(* IEC 61131-3 sources: eCockpitGit/test_project/src/%F%00 Library/%F%JSON/%POU%FB_JSONWriter, 3 files *)

(* ---- %METH%deinitialize.st ---- *)
// |**Version**|**Author**| **Date** |**Changes**
// | 1         | NSN      | 22-06-20 | Creation
METHOD deinitialize

(*%!%__DELIMITER__%!%*)
IF ready THEN
	//Closes up remaining structs
	WHILE treeLevel > 0 DO
		CASE treeTypes[treeLevel] OF
			EStructType.object,EStructType.tArray:
				structEnd();
		END_CASE
	END_WHILE
	bufferPosition			:=		bufferPosition - 1;
	bufferPosition^			:=		EASCII.Null;
	//Initialisation is done
	ready					:=		FALSE;
	//Values are reset
	bufferMaxADR			:=		0;
	inArray					:=		FALSE;
	inObject				:=		FALSE;
	singleVal				:=		FALSE;
	lastComma				:=		0;
	bottomTypeInt			:=		EStructType.none;
	treeLevel				:=		0;
END_IF

(* ---- %METH%initialize.st ---- *)
//This initializes the manager with the correct values
// |**Version**|**Author**| **Date** |**Changes**
// | 1         | NSN      | 22-06-20 | Creation
METHOD initialize : SLMResult
VAR_INPUT
	buffer			:POINTER TO BYTE;	//The address of the file buffer
	bufferSize		:DWORD;				//The size of the file buffer
	singleLine		:BOOL;
	bottomType		:EStructType;
END_VAR
(*%!%__DELIMITER__%!%*)
//Buffer ADR is recorded
IF NOT(ready) THEN
	IF buffer <> 0 AND bufferSize <> 0 THEN
		bufferPosition		:=		buffer;
		bufferAddress		:=		buffer;
		bufferMaxADR		:=		bufferPosition + bufferSize;
		useSingleLine		:=		singleLine;
		bufferInvalid		:=		FALSE;
		//Initialisation is done
		ready				:=		TRUE;
		//First curly bracket is added
		bottomTypeInt		:=		bottomType;
		CASE bottomType OF
			EStructType.object:
				afterKey	:=		TRUE;
				objectStart(singleLine:=FALSE);
			EStructType.tArray:
				afterKey	:=		TRUE;
				arrayStart(singleLine:=FALSE);
		ELSE
			singleVal		:=		TRUE;
		END_CASE
	ELSE
		initialize.success	:=		FALSE;
		initialize.code		:=		ERCodes.FB_JSONWriter_initialize;
		initialize.reason	:=		GTErrors.EmissingInputVars;
	END_IF
ELSE
	initialize.success		:=		FALSE;
	initialize.code			:=		ERCodes.FB_JSONWriter_initialize;
	initialize.reason		:=		GTErrors.EresourceInUse;
END_IF

(* ---- %METH%writeFile.st ---- *)
//This method writes the buffer to a file
// |**Version**|**Author**| **Date** |**Changes**
// | 1         | NSN      | 16-05-21 | Creation
METHOD writeFile
VAR_INPUT
	path			:APath;	//Path of directory to copy from
END_VAR
VAR
	fileResult		:RTS_IEC_RESULT;
	fileHandle		:SysTypes.RTS_IEC_HANDLE;
	lengthBuff		:DWORD;
END_VAR
(*%!%__DELIMITER__%!%*)
fileHandle				:=		SysFile.SysFileOpen(szFile:=path,am:=SysFile.ACCESS_MODE.AM_APPEND_PLUS,pResult:=ADR(fileResult));
IF fileHandle <> 0 AND TO_DWORD(fileHandle) <> 16#FFFFFFFF THEN
	SysFile.SysFileSetPos(hFile:=fileHandle,ulOffset:=0);
	lengthBuff			:=		bufferSize;
	SysFile.SysFileWrite(hFile:=fileHandle,pbyBuffer:=bufferAddress,ulSize:=lengthBuff,pResult:=ADR(fileResult));
	SysFile.SysFileTruncate(hFile:=fileHandle,ulSizeNew:=lengthBuff);
	SysFile.SysFileClose(hFile:=fileHandle);
END_IF
